FUNCTION_BLOCK PUBLIC ABSTRACT FB_Axis
VAR_INPUT
END_VAR
VAR_OUTPUT
	// ================== Axis reference ========================
	Axis				: AXIS_REF;
	
	// ================== State variables =======================
	bError				: BOOL;
	nErrorID			: UDINT;
	bMoves				: BOOL;
	bHaltDone			: BOOL;
	bResetDone			: BOOL;
	bEnableDone			: BOOL;
	bMovePosDone		: BOOL;
END_VAR
VAR
	// ================== Axis function block ===================
	fbMCPower			: MC_Power;
	fbMcReset			: MC_Reset;
	
	// ================== Trigger ================================
	rTrigReset			: R_TRIG;
	
	// ================== Target ================================
	_fVelocity	: LREAL;
	_fPosition	: LREAL;
END_VAR

PROPERTY fPosition : LREAL
GET
fPosition := _fPosition;
END_GET
SET
_fPosition := fPosition;
END_SET
END_PROPERTY

PROPERTY fVelocity : LREAL
GET
fVelocity := _fVelocity;
END_GET
SET
_fVelocity := fVelocity;
END_SET
END_PROPERTY

METHOD PUBLIC ABSTRACT M_Halt : BOOL
VAR_INPUT
	bExecute	:	BOOL;
END_VAR
END_METHOD

METHOD M_Invoke : BOOL
VAR_INPUT
	bEnable		: BOOL;
END_VAR
// ============================================

fbMCPower(	Axis			:= Axis,
			Enable			:= bEnable,
			Enable_Positive	:= bEnable,
			Enable_Negative := bEnable,
			Status			=> bEnableDone);

IF fbMCPower.Error OR Axis.Status.Error THEN
	bError 				:= TRUE;
	nErrorID			:= fbMCPower.ErrorID;
END_IF

Axis.ReadStatus();

bMoves := Axis.Status.Moving;

// ============================================
END_METHOD

METHOD PUBLIC ABSTRACT M_MovePos : BOOL
VAR_INPUT
	bExecute	: BOOL;
END_VAR
END_METHOD

METHOD M_Reset : BOOL
VAR_INPUT
	bExecute	: BOOL;
END_VAR
IF NOT bExecute THEN
	bResetDone		:= FALSE;	
END_IF

rTrigReset(CLK := bExecute);

IF rTrigReset.Q THEN
	bHaltDone		:= FALSE;
	fbMcReset(	Axis	:= Axis,
				Execute	:= TRUE);
ELSE
	fbMcReset(	Axis	:= Axis);
END_IF

// Done / Error
IF fbMcReset.Done OR fbMcReset.Error THEN
	bError			:= fbMcReset.Error;
	nErrorID		:= fbMcReset.ErrorID;
	bResetDone		:= fbMcReset.Done;
	
	fbMcReset(	Axis 	:= Axis,
				Execute	:= FALSE);
END_IF
END_METHOD

END_FUNCTION_BLOCK

(* stored: Version 1.1.0.1, ProductVersion 3.1.4024.6
   POU FB_Axis: Id {ab30e8a8-f177-4a5c-8c2f-acb9e6957c3c}, SpecialFunc None
   Property fPosition: Id {9bab3313-6b0f-4e21-8cc0-bec14d2d6ae2}
   Get Get: Id {629813d0-139e-4120-94ac-4e9dc39ac626}
   Set Set: Id {619cb5fd-4770-474c-a578-cfec2eebfa96}
   Property fVelocity: Id {ffa93d4d-1dcb-45e8-a95a-c597b4b60318}
   Get Get: Id {327edfd0-9486-4068-9066-38c90c543ba0}
   Set Set: Id {f25ee4bc-2b51-47f4-a480-d637ee4910ed}
   Method M_Halt: Id {8a3ef68d-1fdb-41ba-be92-e18639d211fb}
   Method M_Invoke: Id {f82352f2-856c-4aee-bb71-cbcde4291a4d}
   Method M_MovePos: Id {61771372-e1a0-48db-9c1a-e50a26364813}
   Method M_Reset: Id {bc60a92e-a5ce-4ad7-aa94-940a59135b93} *)
